{attribute 'no_explicit_call' := 'This FB is a CLASS and must be accessed using methods or properties'}
{attribute 'enable_dynamic_creation'}
FUNCTION_BLOCK ListForwardEnumerator EXTENDS Disposable IMPLEMENTS I_ForwardEnumerator
VAR
	parent : I_List;
	currentIndex : UDINT;
	invalid : BOOL := FALSE;
	moveNextCalled : BOOL := FALSE;
END_VAR

METHOD FB_init : BOOL
VAR_INPUT
	bInitRetains : BOOL; // if TRUE, the retain variables are initialized (warm start / cold start)
	bInCopyCode : BOOL;  // if TRUE, the instance afterwards gets moved into the copy code (online change)
	List : I_List;
END_VAR
parent := List;
currentIndex := 0;
END_METHOD

PROPERTY PUBLIC IsValid : BOOL
GET
IsValid := (NOT invalid AND parent <> 0);
END_GET
END_PROPERTY

METHOD MoveNext : BOOL
IF invalid OR parent = 0 OR parent.Count = 0 THEN
    RETURN;
END_IF

IF NOT moveNextCalled THEN
	MoveNext := moveNextCalled := TRUE;
	RETURN;
END_IF

IF currentIndex < parent.Count - 1 THEN
    currentIndex := currentIndex + 1;
    MoveNext := TRUE;
END_IF
END_METHOD

METHOD Reset
VAR_INPUT
END_VAR
IF invalid OR parent = 0 THEN
	RETURN;
END_IF

moveNextCalled := FALSE;
currentIndex := 0;
END_METHOD

METHOD PUBLIC TryGet : BOOL
VAR_INPUT
	Destination : ANY;
END_VAR
VAR
	node : I_ListNode;
END_VAR
IF invalid OR parent = 0 OR NOT moveNextCalled THEN
	RETURN;
END_IF

node := parent.Item(currentIndex);

IF node = 0 THEN
	RETURN;
END_IF

TryGet := node.TryGet(Destination);
END_METHOD

METHOD TryGetTo : BOOL
VAR_INPUT
	Destination : PVOID;
	DestinationSize : UDINT;
END_VAR
VAR
	node : I_ListNode;
END_VAR
IF invalid OR parent = 0 OR NOT moveNextCalled THEN
	RETURN;
END_IF

node := parent.Item(currentIndex);

IF node = 0 THEN
	RETURN;
END_IF

TryGetTo := node.TryGetTo(Destination, DestinationSize);
END_METHOD

END_FUNCTION_BLOCK

(* stored: Version 1.1.0.1, ProductVersion 3.1.4024.12
   POU ListForwardEnumerator: Id {71cbcc34-b058-4022-8d0f-92c2cf91e030}, SpecialFunc None
   Folder Constructor: Id {cdeb2947-3a90-4b8f-a836-b2e28e3f7057}
   Method FB_init: Id {561615b3-2102-4e89-85a3-3eb981a30740}
   Property IsValid: Id {0eb1db84-cd2b-4f80-9b94-dc9f9847529f}
   Get Get: Id {7fc3be42-663f-4bd2-bee5-b34cca659a44}
   Method MoveNext: Id {124806d4-b465-483c-825d-a72774a6ff60}
   Method Reset: Id {f422f349-f379-43b1-b232-77cd4258d20c}
   Method TryGet: Id {fc9b3816-84f5-4733-83b3-f353243e6fb9}
   Method TryGetTo: Id {c779c4e7-cbea-4286-b465-4d39f43aee99} *)
